INTERFACE ITF_MotorZuigSchuif

PROPERTY Status : E_MotorZuigSchuifStatus
GET
END_GET
SET
END_SET
END_PROPERTY

METHOD SturingKort : BOOL
VAR_INPUT
END_VAR
END_METHOD

METHOD SturingLang : BOOL
VAR_INPUT
END_VAR
END_METHOD

END_INTERFACE

(* stored: Version 1.1.0.1
   Itf ITF_MotorZuigSchuif: Id {f9748cdf-06f5-4267-9c6d-e50a2c3d724e}
   Property Status: Id {f0a59b0b-852a-4a5c-ad39-ecc3f0017762}
   Get Get: Id {d595cb8c-9f7d-4041-8f43-d698461fb38e}
   Set Set: Id {1b61f6cb-ab1f-4b7e-acf5-7370a7c268f8}
   Method SturingKort: Id {647bc108-0a5b-4ab4-a48e-be644f3e59f7}
   Method SturingLang: Id {a9d25a77-3eaf-4bc2-9cdb-424a246396e5} *)
